RoboDK station: RobotPhoto.rdk

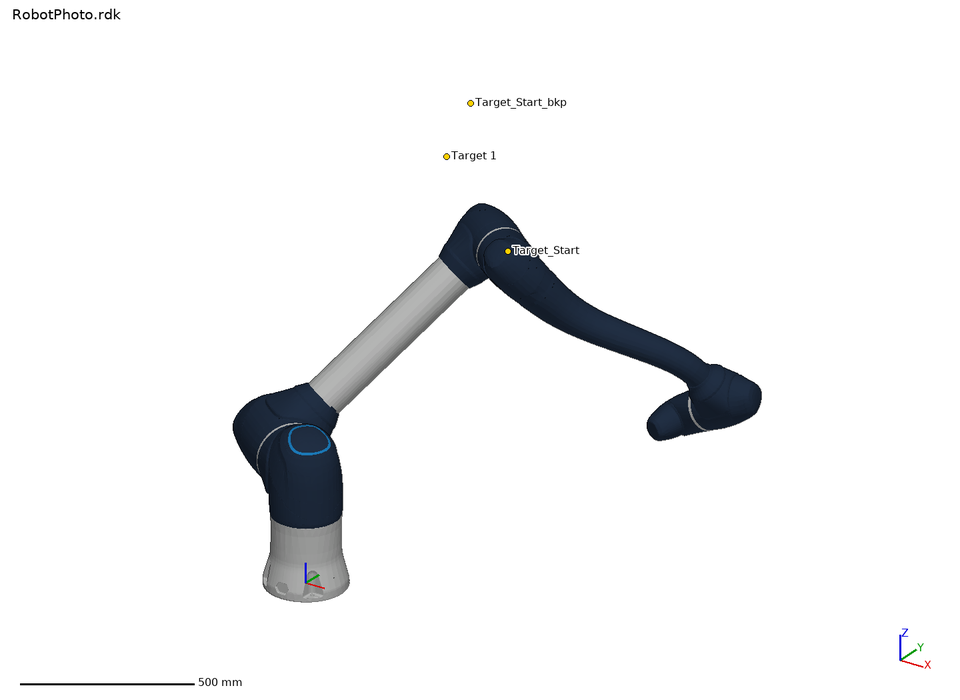
[picture v0: the station drawn from its stored meshes, robots at their saved joint values, targets as dots, program paths as lines]
Station RobotPhoto (saved by RoboDK 5.5.1). Poses are relative to the parent item; angles as X-Y-Z fixed-axis rotations.
  - frame Doosan Robotics H2017 Base at (0, 0, 0) mm
    - robot Doosan Robotics H2017: 6 axes, payload 20 kg, reach 1700 mm, repeatability 0.1 mm
        modified DH rows (alpha deg, a mm, theta deg, d mm): 0, 0, 180, 344.3; -90, 0, -90, -9.9; 0, 845, -90, 0; -90, 0, 0, 734; 90, 0, 0, 0; -90, 0, 180, 121
        joint limits [-360, -130, -160, -360, -360, -360] to [360, 130, 160, 360, 360, 360]; home [0, 0, -90, 0, 0, 0]; saved at [54.31, 49.543, 88.58, -224.921, 57.286, 208.113]
    - target Target_Start (Cartesian target) at (-23.69, 1046.9, 635.51) mm, rotated rx -177.88 ry 89.73 rz -87.12 deg; joints [90.754, 25.463, 104.469, -0.009, -39.662, -0.003] of Doosan Robotics H2017
    - target Target_Start_bkp (Cartesian target) at (-21.25, 855.52, 1185.27) mm, rotated rx -177.88 ry 89.73 rz -87.12 deg; joints [90.76, 0.05, 90.22, -0.01, 0, 0] of Doosan Robotics H2017
    - target Target 1 (Cartesian target) at (-19.64, 733.98, 1064.97) mm, rotated rx -180 ry -0.26 rz -89.24 deg; joints [90.76, 0.05, 90.21, 0, 90, 0] of Doosan Robotics H2017
  - Python program Prog1 (listed below)

--- Python program Prog1 ---
longueur, hauteur = 1500, 700  # Taille du rectange à analyser [mm]

LONGUEUR_FOTO = 150  # Longueur prise par la caméra [mm] quand elle est à DIST_CAM
HAUTEUR_FOTO = 120  # Hauteur prise par la caméra [mm] quand elle est à DIST_CAM

from robodk import robolink    # RoboDK API
from robodk import robomath    # Robot toolbox

from robodk import *      # RoboDK API
from robolink import *    # Robot toolbox

from math import *
from time import sleep

from LaBrise.take_picture import image_viewer

os.system('cls')
cam = image_viewer()

#---[CONNEXION]---#
RDK = Robolink()
robot = RDK.ItemUserPick('Select a robot', ITEM_TYPE_ROBOT)
if not robot.Valid():
    raise Exception('No robot selected or available')
'''
RDK = Robolink()

robot = RDK.ItemUserPick('Select a robot', ITEM_TYPE_ROBOT)
if not robot.Valid():
    raise Exception('No robot selected or available')

RUN_ON_ROBOT = True

if RDK.RunMode() != RUNMODE_SIMULATE:
    RUN_ON_ROBOT = False

if RUN_ON_ROBOT:
    success = robot.Connect()
    status, status_msg = robot.ConnectedState()
    if status != ROBOTCOM_READY:
        print(status_msg)
        raise Exception("Failed to connect: " + status_msg)

    RDK.setRunMode(RUNMODE_RUN_ROBOT)'''
#-----------------#

joints_ref = robot.Joints()

robot.MoveJ(RDK.Item('Target 1').Pose())

start_pose = RDK.Item('Target_Start').Pose()
robot.MoveJ(start_pose)

robot.setPoseFrame(robot.PoseFrame())
robot.setPoseTool(robot.PoseTool())

robot.setZoneData(10)
robot.setSpeed(50,5)

#---[CALCUL DU GRID]---#
num_grid_x = ceil(longueur/LONGUEUR_FOTO)
overlapping_x = (num_grid_x*LONGUEUR_FOTO - longueur)/(num_grid_x-1)
grid_x = [(LONGUEUR_FOTO/2)-(longueur/2) + i*(LONGUEUR_FOTO-overlapping_x) for i in range(num_grid_x)]

num_grid_y = ceil(hauteur/HAUTEUR_FOTO)
overlapping_y = (num_grid_y*HAUTEUR_FOTO - hauteur)/(num_grid_y-1)
grid_y = [(HAUTEUR_FOTO/2)-(hauteur/2) + i*(HAUTEUR_FOTO-overlapping_y) for i in range(num_grid_y)]

grid = []
for y in range(num_grid_y):
    for x in range(num_grid_x):
        if y%2 == 0:
            grid.append((grid_x[x], grid_y[-y-1]))
        else:
            grid.append((grid_x[-x-1], grid_y[-y-1]))
#----------------------#

counter = 0
for point in grid:
    target = Mat(start_pose)
    pos = target.Pos()
    pos[2] += point[1]
    pos[0] -= point[0]
    target.setPos(pos)

    robot.MoveJ(target)

    cam.take_picture(sys.argv, str(counter) + '.png')

    sleep(1)
    counter += 1
